// TIA Portal project "queueOfItemsRevised" (V17)

(* hardware
DEVICE "S71500/ET200MP-Station_1"  S7-1500 station
   slot 0: "Profilschiene_0"  6ES7 590-1***0-0AA0
   slot 1: "PLC_1"  CPU 1511-1 PN  6ES7 511-1AK00-0AB0  V1.8
   slot 2: "AI 8xU/I/RTD/TC ST_1"  AI 8xU/I/RTD/TC ST  6ES7 531-7KF00-0AB0  V2.0
   slot 3: "AI 8xU/I/RTD/TC ST_2"  AI 8xU/I/RTD/TC ST  6ES7 531-7KF00-0AB0  V2.0
   slot 4: "AI 8xU/I/RTD/TC ST_3"  AI 8xU/I/RTD/TC ST  6ES7 531-7KF00-0AB0  V2.0
   slot 5: "AI 8xU/I/RTD/TC ST_4"  AI 8xU/I/RTD/TC ST  6ES7 531-7KF00-0AB0  V2.0
   slot 6: "DI 16x24VDC BA_1"  DI 16x24VDC BA  6ES7 521-1BH10-0AA0  V1.0
*)

// ===== PLC "PLC_1"  CPU 1511-1 PN =====

VAR_GLOBAL   // PLC tag table "Standard-Variablentabelle"
   "Item Ready" AT %E0.0 : Bool;
   "At Entry" AT %I0.1 : Bool;
   "At Exit" AT %I0.2 : Bool;
   "Entry Conveyor" AT %Q0.0 : Bool;
   "Buffer Conveyor" AT %Q0.1 : Bool;
   "Tag_1" AT %M0.0 : Bool;
   "threeCountMemory" AT %M0.1 : Bool;
   "secondCounterMemory" AT %M0.2 : Bool;
   "Tag_2" AT %M0.3 : Bool;
   "bufferConveyorActivate" AT %M0.5 : Bool;
   "bufferConveyor2Activate" AT %M0.6 : Bool;
END_VAR

// folder: System blocks/Program resources

DATA_BLOCK "box counter"   // DB1
{ S7_Optimized_Access := 'TRUE' }
AUTHOR : Simatic
FAMILY : IEC
NAME : CNTR
VERSION : 1.0
// stored: InstanceOfName IEC_COUNTER
"IEC_COUNTER"
BEGIN
END_DATA_BLOCK

DATA_BLOCK "second counter"   // DB2
{ S7_Optimized_Access := 'TRUE' }
AUTHOR : Simatic
FAMILY : IEC
NAME : CNTR
VERSION : 1.0
// stored: InstanceOfName IEC_COUNTER
"IEC_COUNTER"
BEGIN
END_DATA_BLOCK

// folder: (top level)

FUNCTION "MHJ-PLC-Lab-Function-S71500" : Void   // FC9000, SCL
{ S7_Optimized_Access := 'TRUE' }
VERSION : 0.1
   VAR_TEMP
      Value : Byte;
      ForCounter : Int;
   END_VAR
   VAR CONSTANT
      Value_01_DW : DWord := 16#1223_5486;
      Value_02_DW : DWord := 16#A6C9_D1F5;
   END_VAR
BEGIN

   #Value:=PEEK(area := 16#82,
        dbNumber := 0,
        byteOffset := 511);
   #Value := #Value + 1;

   POKE(area := 16#82,
        dbNumber := 0,
        byteOffset := 511,
        value := #Value);

   POKE(area := 16#82,
        dbNumber := 0,
        byteOffset := 1016,
        value := #Value_01_DW);
   POKE(area := 16#82,
        dbNumber := 0,
        byteOffset := 1020,
        value := #Value_02_DW);

   FOR #ForCounter := 0 TO 63 DO
       #Value:=PEEK(area := 16#1,
            dbNumber := 0,
            byteOffset := #ForCounter);
       POKE(area := 16#81,
            dbNumber := 0,
            byteOffset := #ForCounter,
            value := #Value);
   END_FOR;
   #Value := PEEK(area := 16#1,
                  dbNumber := 0,
                  byteOffset := 512);
   POKE(area := 16#82,
        dbNumber := 0,
        byteOffset := 512,
        value := #Value);
END_FUNCTION

ORGANIZATION_BLOCK "Main"   // OB1, LAD, ProgramCycle
TITLE = "Main Program Sweep (Cycle)"
{ S7_Optimized_Access := 'TRUE' }
VERSION : 0.1
   VAR_INPUT
      Initial_Call : Bool;   // Initial call of this OB
      Remanence : Bool;   // =True, if remanent data are available
   END_VAR
   VAR_TEMP   // added for the SCL form of the ladder/FBD networks
      _w1 : Bool;
   END_VAR
BEGIN

REGION Network 1
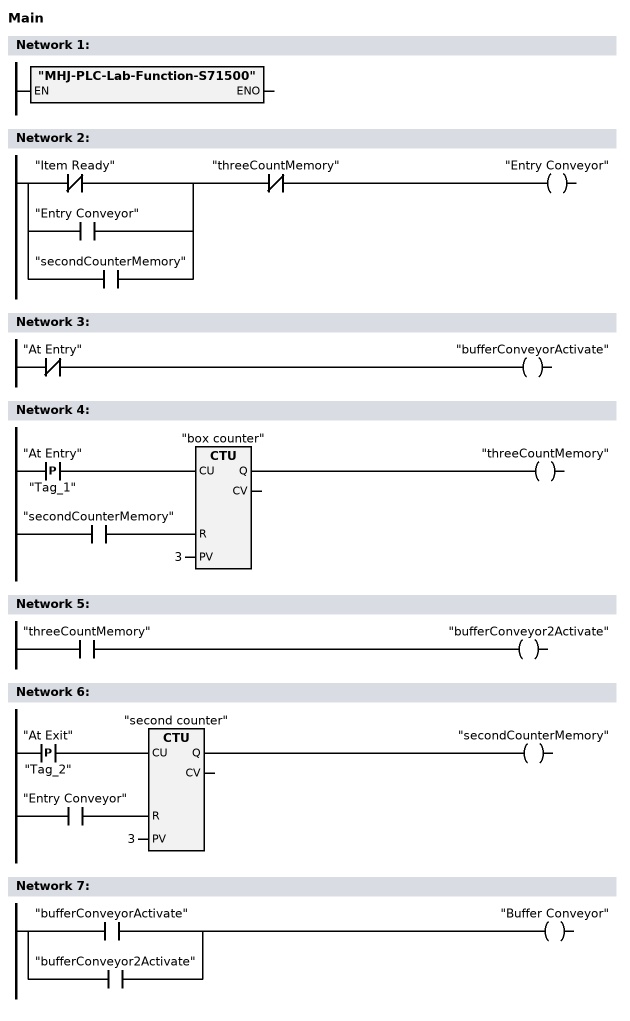
   RUNG wire#powerrail
      "MHJ-PLC-Lab-Function-S71500"()
   END_RUNG
   // the same network as SCL:
   "MHJ-PLC-Lab-Function-S71500"();
END_REGION

REGION Network 2
   RUNG wire#powerrail
      I_Contact( "Item Ready" )
      wire#w1
      I_Contact( "threeCountMemory" )
      Coil( "Entry Conveyor" )
   END_RUNG
   RUNG wire#powerrail
      Contact( "Entry Conveyor" )
   END_RUNG wire#w1
   RUNG wire#powerrail
      Contact( "secondCounterMemory" )
   END_RUNG wire#w1
   // the same network as SCL:
   "Entry Conveyor" := (NOT "Item Ready" OR "Entry Conveyor" OR "secondCounterMemory") AND NOT "threeCountMemory";
END_REGION

REGION Network 3
   RUNG wire#powerrail
      I_Contact( "At Entry" )
      Coil( "bufferConveyorActivate" )
   END_RUNG
   // the same network as SCL:
   "bufferConveyorActivate" := NOT "At Entry";
END_REGION

REGION Network 4
   #_w1 := "At Entry" AND NOT "Tag_1";   // rising edge of "At Entry"
   "Tag_1" := "At Entry";
   "box counter".CTU(CU := #_w1, R := "secondCounterMemory", PV := 3);
   "threeCountMemory" := "box counter".Q;
END_REGION

REGION Network 5
   RUNG wire#powerrail
      Contact( "threeCountMemory" )
      Coil( "bufferConveyor2Activate" )
   END_RUNG
   // the same network as SCL:
   "bufferConveyor2Activate" := "threeCountMemory";
END_REGION

REGION Network 6
   #_w1 := "At Exit" AND NOT "Tag_2";   // rising edge of "At Exit"
   "Tag_2" := "At Exit";
   "second counter".CTU(CU := #_w1, R := "Entry Conveyor", PV := 3);
   "secondCounterMemory" := "second counter".Q;
END_REGION

REGION Network 7
   RUNG wire#powerrail
      Contact( "bufferConveyorActivate" )
      wire#w1
      Coil( "Buffer Conveyor" )
   END_RUNG
   RUNG wire#powerrail
      Contact( "bufferConveyor2Activate" )
   END_RUNG wire#w1
   // the same network as SCL:
   "Buffer Conveyor" := "bufferConveyorActivate" OR "bufferConveyor2Activate";
END_REGION
END_ORGANIZATION_BLOCK